INTERFACE I_RaDecTelescope EXTENDS I_Telescope

PROPERTY DeclinationOffset : LREAL
GET
END_GET
SET
END_SET
END_PROPERTY

PROPERTY HourAngleOffset : LREAL
GET
END_GET
SET
END_SET
END_PROPERTY

END_INTERFACE

(* stored: Version 1.1.0.1, ProductVersion 3.1.4024.15
   Itf I_RaDecTelescope: Id {fca915a4-38d8-47a2-9bf5-dd2cdf97023e}
   Property DeclinationOffset: Id {a730f447-9940-48ab-863f-161dd001843d}
   Get Get: Id {56007fc8-4474-49ec-bf47-d026a049fd60}
   Set Set: Id {0358f7e9-95c3-4de1-8d50-74d0235aa117}
   Property HourAngleOffset: Id {777dfd7c-8617-4f6a-b2b2-7aaf194d6ef0}
   Get Get: Id {5686a4a6-92a0-4f61-9de3-93dbb226119a}
   Set Set: Id {eefa9c79-1d73-4bf1-be58-dce6831cf612} *)
